FUNCTION_BLOCK CL_AxisL2RighFront EXTENDS CL_AxisRobot
var
END_VAR

SUPER^();

METHOD PROTECTED InitDefect : BOOL
sWhichAxis := 'right(L2)-front';
InitDefect := true;
END_METHOD

END_FUNCTION_BLOCK

(* stored: Version 1.1.0.1, ProductVersion 3.1.4024.12
   POU CL_AxisL2RighFront: Id {6a3d2686-b758-4c65-905f-34cb410c5611}, SpecialFunc None
   Method InitDefect: Id {a3c088b0-c881-48fa-a2f2-a087f1582cf9} *)
